// TIA Portal V20 export
// export: Created 2026-07-10T11:12:28.6019688Z, ExportSetting WithDefaults, DisplayName Totally Integrated Automation Portal, DisplayVersion V20, DisplayName TIA Portal Openness, DisplayVersion V20, DisplayName TIA Portal Version Control Interface, DisplayVersion V20, DisplayName STEP 7 Professional, DisplayVersion V20, DisplayName STEP 7 Safety, DisplayVersion V20, DisplayName WinCC Basic/Comfort/Advanced, DisplayVersion V20, DisplayName WinCC Unified, DisplayVersion V20
FUNCTION_BLOCK "FlowCounter"   // FB27, SCL
{ S7_Optimized_Access := 'TRUE' }
VERSION : 0.1
// stored: AutoNumber true, IsIECCheckEnabled false, IsRetainMemResEnabled false, MemoryReserve 100, SetENOAutomatically false, UDAEnableTagReadback false
   VAR_IN_OUT
      Pulse : Bool;
      DailyCount : DInt;
      TotalCount : DInt;
      PulseWeight : Real;
      Consumption : Real;
      DailyValue : Real;
      TotalValue : Real;
   END_VAR
   VAR
      R_TRIG_Instance { S7_SetPoint := 'True'} : R_TRIG;
      HourTimer { S7_SetPoint := 'True'} : TON_TIME;
      PrevValue { S7_SetPoint := 'True'} : Real;
      TimeNow : DTL;
      TimeLast : DTL;
      Ret : Int;
      TimeDif : Time;
      FilterArr : Array[0..3] of Real;
      i : Int;
      NoFlowTON { S7_SetPoint := 'True'} : TON_TIME;
   END_VAR
   VAR_TEMP
      j : Int;
      sum : Real;
   END_VAR
BEGIN
   #R_TRIG_Instance(CLK := #Pulse,
                    Q => #R_TRIG_Instance.Q);

   #HourTimer.TON(IN := TRUE,
   PT := T#3600s);

   #NoFlowTON(IN := TRUE,
              PT := T#300s);

   IF #R_TRIG_Instance.Q THEN
       RESET_TIMER(#NoFlowTON);
       #R_TRIG_Instance.CLK := FALSE;
       IF (#i > 3) THEN
           #i := 0;
       END_IF;

       #DailyCount += 1;
       #TotalCount += 1;
       #Ret := RD_SYS_T(#TimeNow);
       #TimeDif := #TimeNow - #TimeLast;
       #FilterArr[#i] := 3600 * 1000 / DINT_TO_REAL(#TimeDif) * #PulseWeight;
       FOR #j := 0 TO 3 DO
           #sum += #FilterArr[#j];
       END_FOR;

       #Consumption := #sum / 4;
       #TimeLast := #TimeNow;
       #i += 1;
       #sum := 0;

   END_IF;

   #DailyValue := UDINT_TO_REAL(#DailyCount) * #PulseWeight;
   #TotalValue := UDINT_TO_REAL(#TotalCount) * #PulseWeight;

   IF #NoFlowTON.Q THEN
       #Consumption := 0;
   END_IF;

   IF "Config".HMI_ResetWaterCounter THEN
       #DailyCount := 0;
       #TotalCount := 0;
   END_IF;
END_FUNCTION_BLOCK
